(* PLC project M3_13, Desconocido M3_13 1 *)
(* stored: creationDateTime 2025-05-15T11:40:54, modificationDateTime 2025-06-10T00:04:41 *)

PROGRAM Main
  VAR
    xMarcha : BOOL;  (* Marcha de la bomba principal *)
    xParada : BOOL;  (* Parada de la bomba principal *)
    xBomba : BOOL;  (* Bomba principal *)
    xFalla : BOOL;  (* Falla de la Bomba *)
    xAlertaFalla : BOOL;  (* Alerta de Falla de la Bomba *)
    TON0 : TON;
    TON1 : TON;
    CTU0 : CTU;
  END_VAR
  VAR  (* added by the conversion: wires and edge detectors of the diagram *)
    R_TRIG1 : R_TRIG;
  END_VAR

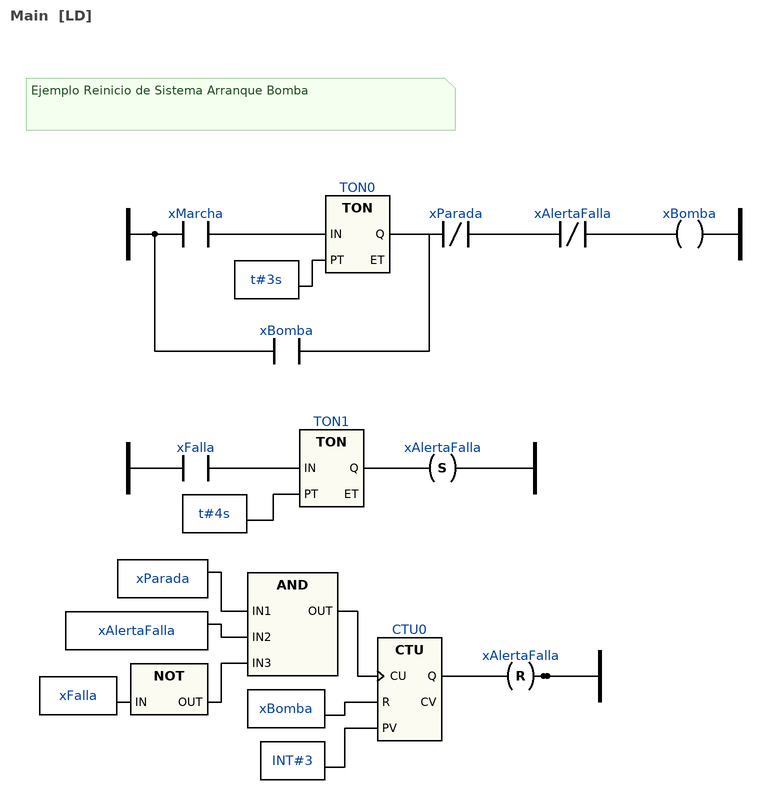
(* LD diagram, written out as Structured Text *)
(* Ejemplo Reinicio de Sistema Arranque Bomba *)
TON0(IN := xMarcha, PT := t#3s);
xBomba := (xBomba OR TON0.Q) AND NOT xParada AND NOT xAlertaFalla;
TON1(IN := xFalla, PT := t#4s);
IF TON1.Q THEN xAlertaFalla := TRUE; END_IF;
R_TRIG1(CLK := xParada AND xAlertaFalla AND NOT xFalla);
CTU0(CU := R_TRIG1.Q, R := xBomba, PV := INT#3);
IF CTU0.Q THEN xAlertaFalla := FALSE; END_IF;
END_PROGRAM

CONFIGURATION Config0
  RESOURCE Res0 ON PLC
    TASK task0(INTERVAL := T#20ms, PRIORITY := 0);
    PROGRAM instance0 WITH task0 : Main;
  END_RESOURCE
END_CONFIGURATION
